// TIA Portal V17 export
// export: Created 2025-03-05T08:02:32.7444535Z, ExportSetting WithDefaults, DisplayName Totally Integrated Automation Portal, DisplayVersion V17 Update 8, DisplayName TIA Portal Openness, DisplayVersion V17 Update 8, DisplayName TIA Portal Version Control Interface, DisplayVersion V17, DisplayName SINAMICS Startdrive Advanced, DisplayVersion V17 SP2, DisplayName SINAMICS Startdrive G110M, G120, G120C, G120D, G120P, G115D, DisplayVersion V17 SP2, DisplayName SINAMICS Startdrive G130, G150, S120, S150, SINAMICS MV, S210, DisplayVersion V17 SP2, DisplayName STEP 7 Professional, DisplayVersion V17 Update 8, DisplayName SINUMERIK ONE STEP 7 Toolbox, DisplayVersion V17 Update 12, DisplayName SINUMERIK 840D sl STEP 7 Toolbox, DisplayVersion V17 Update 12, DisplayName STEP 7 Safety, DisplayVersion V17 Update 6, DisplayName WinCC Advanced, DisplayVersion V17 Update 8
TYPE "U03_MEAS_STATION_FACE_A.U03_FACE_A_MEAS_Read"
// stored: IsFailsafeCompliant false
   STRUCT
      Status { ExternalWritable := 'False'} : Int;
      ProfilerConfiguration { ExternalWritable := 'False'} : Bool;
      AnalyzerConfiguration { ExternalWritable := 'False'} : Bool;
      DMCStructure { ExternalWritable := 'False'} : Bool;
      Acquisition { ExternalWritable := 'False'} : Bool;
      ProfilerInitialization { ExternalWritable := 'False'} : Bool;
      UmbrellaAnalysis { ExternalWritable := 'False'} : Bool;
      RunOutAnalysis { ExternalWritable := 'False'} : Bool;
      DistanceCalculation { ExternalWritable := 'False'} : Bool;
      SurfaceDefectsAnalysis { ExternalWritable := 'False'} : Bool;
      StorageError { ExternalWritable := 'False'} : Bool;
      DatabaseConnection { ExternalWritable := 'False'} : Bool;
      SensorTemperature { ExternalWritable := 'False'} : Real;
      "Status Fixture 1" { ExternalWritable := 'False'} : Bool;
   END_STRUCT;
END_TYPE
